FUNCTION_BLOCK FB_RealToBytes // Convert Real data into 4 bytes
VAR_INPUT
	IN_DATA : REAL; //The Input Data in Real Data type 
END_VAR
VAR_OUTPUT
	UpperByteA :BYTE; //  UpperByte 1 the 25-32 bits from the Data word (Count from Right) 
	UpperByteB :BYTE; //  UpperByte 2 the 17-24 bits from the Data word (Count from Right)
	LowerByteC :BYTE; //  LowerByte 1 the 9-16 bits from the Data word (Count from Right)
	LowerByteD :BYTE; //  LowerByte 2 the 1-8 bits from the Data word (Count from Right)
END_VAR
VAR
	b_Input : BYTE;
	w_Input : DWORD;
	r_Data 	: REAL;
	w_Input1: WORD;
	UpperDWord : DWORD;
	LowerDWord : DWORD;
	
	UpperWord: WORD;
	LowerWord: WORD;
	
	UpperWordA: WORD;
	UpperWordB: WORD;
	LowerWordA: WORD;
	LowerWordB: WORD;
END_VAR

r_Data :=  IN_DATA *1000; // remove decimal from real
w_Input:= TO_DWORD(r_Data);  // Change from real to word

// DWORD DATA Split into two DWORD 
UpperDWord := SHR(w_Input,16);
LowerDWord := w_Input - SHL(UpperDWord,16);

//  Change into WORD
UpperWord := TO_WORD(UpperDWord);
LowerWord := TO_WORD(LowerDWord);

// Convert WORD to Byte Calculation
UpperWordA := SHR(UpperWord,8);
UpperWordB := UpperWord - SHL(UpperWordA,8);

LowerWordA := SHR(LowerWord,8);
LowerWordB := LowerWord - SHL(LowerWordA,8);

//  Change into Byte
UpperByteA	:= TO_BYTE(UpperWordB);
UpperByteB	:= TO_BYTE(UpperWordA);

LowerByteC	:= TO_BYTE(LowerWordB);
LowerByteD	:= TO_BYTE(LowerWordA);

END_FUNCTION_BLOCK

(* stored: Version 1.1.0.1, ProductVersion 3.1.4024.11
   POU FB_RealToBytes: Id {a8a83422-7963-4444-baad-8c648823c227}, SpecialFunc None *)
